TYPE ST_SCANNER_HoneywellStatus :
STRUCT
	bStringReceived			: BOOL;
	bExtStringReceived			: BOOL;
	bHandScanerPortOK			: BOOL;
	bHandScannerBaudrateOK	: BOOL;
	sLastScannerBarcode		: STRING(255);
END_STRUCT
END_TYPE

(* stored: Version 1.1.0.1, ProductVersion 3.1.4024.15
   DUT ST_SCANNER_HoneywellStatus: Id {99c02ef8-273b-4e2e-bce7-6bdb0dee2e5e} *)
